// Mitsubishi GX Works2 project: 세탁기능   PLC: Q03UDV

PROGRAM MAIN
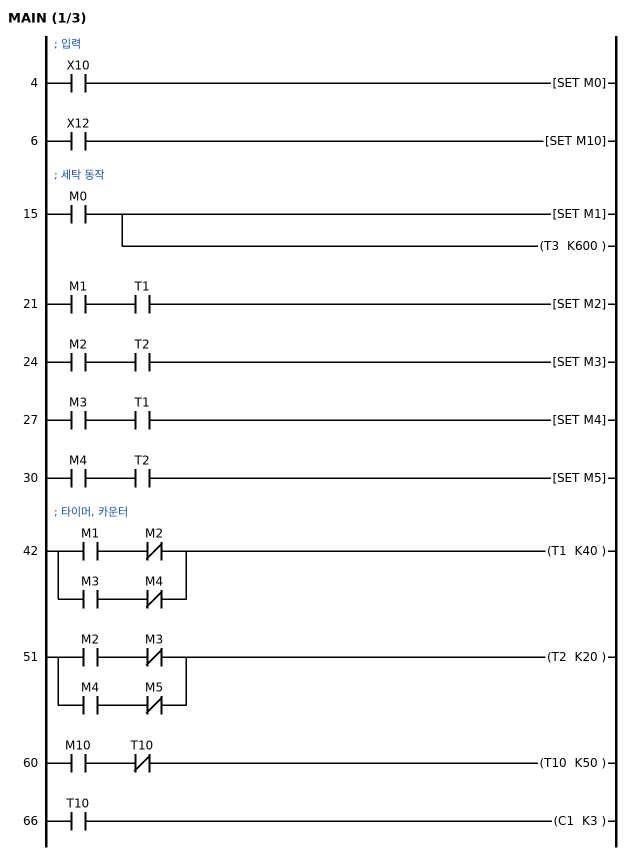
; 입력
4     LD      X10
      SET     M0
6     LD      X12
      SET     M10
; 세탁 동작
15    LD      M0
      SET     M1
      OUT     T3 K600
21    LD      M1
      AND     T1
      SET     M2
24    LD      M2
      AND     T2
      SET     M3
27    LD      M3
      AND     T1
      SET     M4
30    LD      M4
      AND     T2
      SET     M5
; 타이머, 카운터
42    LD      M1
      ANI     M2
      LD      M3
      ANI     M4
      ORB
      OUT     T1 K40
51    LD      M2
      ANI     M3
      LD      M4
      ANI     M5
      ORB
      OUT     T2 K20
60    LD      M10
      ANI     T10
      OUT     T10 K50
66    LD      T10
      OUT     C1 K3
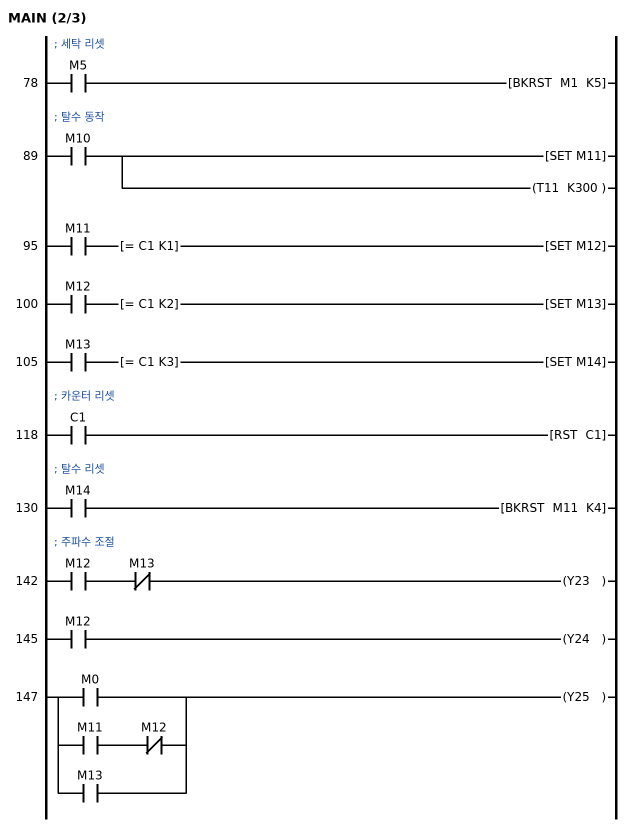
; 세탁 리셋
78    LD      M5
      BKRST   M1 K5
; 탈수 동작
89    LD      M10
      SET     M11
      OUT     T11 K300
95    LD      M11
      AND=    C1 K1
      SET     M12
100   LD      M12
      AND=    C1 K2
      SET     M13
105   LD      M13
      AND=    C1 K3
      SET     M14
; 카운터 리셋
118   LD      C1
      RST     C1
; 탈수 리셋
130   LD      M14
      BKRST   M11 K4
; 주파수 조절
142   LD      M12
      ANI     M13
      OUT     Y23
145   LD      M12
      OUT     Y24
147   LD      M0
      LD      M11
      ANI     M12
      ORB
      OR      M13
      OUT     Y25
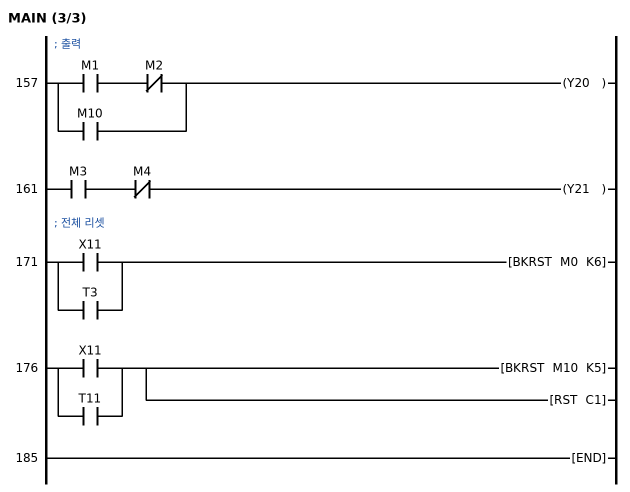
; 출력
157   LD      M1
      ANI     M2
      OR      M10
      OUT     Y20
161   LD      M3
      ANI     M4
      OUT     Y21
; 전체 리셋
171   LD      X11
      OR      T3
      BKRST   M0 K6
176   LD      X11
      OR      T11
      BKRST   M10 K5
      RST     C1
185   END
END_PROGRAM
